Staubli VAL3: consume.pgx

program consume(num& x_nStatus (dimensions=1), num x_nReference (dimensions=1))
  local num l_nConnStatus
  local num l_nData[4]
  local num l_nValue
  local num l_nBinaryStatus
begin
  // consumes 4 bytes and verifes with the reference
  // does nothing if first return parameter is not 0
  // return
  //    -2 - timeout
  //    -1 - unexpected value
  //     0 - expected value
  if x_nStatus<0
    return
  endIf
  x_nStatus=-1
  l_nConnStatus=sioGet(siConn,l_nData)
  if l_nConnStatus==4
    l_nBinaryStatus=fromBinary(l_nData,4,"4l",l_nValue)
    if l_nData==x_nReference and l_nBinaryStatus==1
      x_nStatus=0
    endIf
  elseIf l_nConnStatus==-1
    x_nStatus=-2
  endIf
end
